// TIA Portal V18 export
VAR_GLOBAL   // PLC tag table "Outputs"
   "Left Driver On/Off" AT %Q0.0 : Bool;
   "Left Driver Reversing" AT %Q0.1 : Bool;
   "Left Driver Fault" AT %Q0.2 : Bool;
   "Left Driver DI4 STO" AT %Q0.3 : Bool;
   "Left Driver DI5 STO" AT %Q0.4 : Bool;
   "Right Driver On/Off" AT %Q0.5 : Bool;
   "Right Driver Reversing" AT %Q0.6 : Bool;
   "Right Driver Fault" AT %Q0.7 : Bool;
   "Right Driver DI4 STO" AT %Q1.0 : Bool;
   "Right Driver DI5 STO" AT %Q1.1 : Bool;
   "Cab Driver On/Off" AT %Q2.0 : Bool;
   "Cab Driver Reversing" AT %Q2.1 : Bool;
   "Cab Driver Fault Reset" AT %Q2.2 : Bool;
   "Cab Driver DI4 STO" AT %Q2.3 : Bool;
   "Cab Driver DI5 STO" AT %Q2.4 : Bool;
   "MC - Main Contactor" AT %Q3.0 : Bool;
   "C1 - Hydraulic" AT %Q3.1 : Bool;   // MC-105, MC-106, MC-107, MC-108, Cable No:200, MKS2
   "C2 - Hose power" AT %Q3.2 : Bool;
   "C3 - Tunnel Lights" AT %Q3.3 : Bool;
   "C4 - Tunnel Lights UPS" AT %Q3.4 : Bool;
   "C5 - Ext Lighting" AT %Q3.5 : Bool;
   "R2 - Bumper Red Light iptal" AT %Q3.7 : Bool;
   "R1 - SafetyEdge Red Light" AT %Q3.6 : Bool;   // MC-256 MC-257 MC-258, Cable No:204, F11
   "R4 - Mania Lights" AT %Q4.1 : Bool;
   "R6 - Cab Warning Light & Buzzer" AT %Q4.3 : Bool;
   "R7 - Motor Brake Left" AT %Q4.4 : Bool;
   "R8 - Motor Brake Right" AT %Q4.5 : Bool;
   "R12 - Valve Up" AT %Q5.1 : Bool;
   "R13 - Valve Down" AT %Q5.2 : Bool;
   "R14 - Valve Em Down" AT %Q5.3 : Bool;
   "R15 - Valve V4 & V5 Columns Down" AT %Q5.4 : Bool;
   "R3 - Left & Right Warning Lights" AT %Q4.0 : Bool;
   "R9 - Cabin Motor Brake" AT %Q4.6 : Bool;
   "R20 - PBB On" AT %Q5.5 : Bool;
   "R21 - PBB Error/Fault/Alarm" AT %Q5.6 : Bool;
   "R22 - Autoleveller On" AT %Q5.7 : Bool;
   "R23 - AutoLeveller Fault" AT %Q6.0 : Bool;
   "R24 - SafetyShoe Activated" AT %Q6.1 : Bool;
   "R25 - Fire Detector" AT %Q6.2 : Bool;
   "R50 - HMI Power" AT %Q10.0 : Bool;
   "R51 - SafetyShoe Power" AT %Q10.1 : Bool;
   "C52 - Left Canopy FW" AT %Q10.6 : Bool;
   "C53 - Left Canopy BW" AT %Q10.7 : Bool;
   "C54 - Right Canopy FW" AT %Q11.0 : Bool;
   "C55 - Right Canopy BW" AT %Q11.1 : Bool;
   "C50 - Cab Floor FW" AT %Q10.4 : Bool;
   "C51 - Cab Floor BW" AT %Q10.5 : Bool;
   "C56 - AutoLeveller FW" AT %Q11.2 : Bool;
   "C57 - AutoLeveller BW" AT %Q11.3 : Bool;
   "CP - Buzzer" AT %Q12.0 : Bool;
   "CP - Alarm Red Light" AT %Q12.1 : Bool;
   "CP - PBB Start Green Light" AT %Q12.2 : Bool;
   "CP - Reset Red Light" AT %Q12.3 : Bool;
   "CP - Button Int Lighting Light" AT %Q12.4 : Bool;
   "CP - Button Ext Lighting Light" AT %Q12.5 : Bool;
   "CP - Button Em Stop Light" AT %Q12.7 : Bool;
   "PCA Active OUT" AT %Q13.2 : Bool;
   "GPU1 Active OUT" AT %Q13.3 : Bool;
   "GPU2 Active OUT" AT %Q13.4 : Bool;
   "PBB HOME" AT %Q13.0 : Bool;
   "PBB Autoleveler ON" AT %Q13.1 : Bool;
END_VAR
